(* IEC 61131-3 sources: POMIRTS_lab3/AS/Library/AsETH, 3 files *)

(* ---- AsETH.typ ---- *)
(********************************************************************
 * COPYRIGHT -- Bernecker + Rainer
 ********************************************************************
 * Library: AsEth
 * File: AsEth.typ
 * Author: B+R
 ********************************************************************
 * Data types of library AsEth
 ********************************************************************)

TYPE
    ethSTATISTICS_typ	: STRUCT				(*statistics*)
		bytesrecv		: UDINT;				(*bytes received*)
		bytessend		: UDINT;				(*bytes sent*)
		packetsrecv		: UDINT;				(*packets received*)
		packetssend		: UDINT;				(*packets send*)
		mcpacketsrecv	: UDINT;				(*multicast packets received*)
		mcpacketssend	: UDINT;				(*multicats packets sent*)
		errorrecv		: UDINT;				(*input errors*)
		errorsend		: UDINT;				(*output errors*)
		errorframe		: UDINT;				(*frame errors*)
		errorcrc		: UDINT;				(*crc errors*)
		collisions		: UDINT;				(*collisions*)
		latecollision	: UDINT;				(*late collisions*)
		drops			: UDINT;				(*dropped on input*)
		lostcarrier		: UDINT;				(*lost carrier*)
		underflow		: UDINT;				(*silo underflow*)
		retry			: UDINT;				(*retries after 16 collisions*)
		noproto			: UDINT;				(*destined for unsupported protocol*)
		intrecv			: UDINT;				(*reveive interrupts*)
		intsend			: UDINT;				(*transmit interrupts*)
		bufferrecv		: UDINT;				(*receive buffer errror*)
		buffersend		: UDINT;				(*send buffer errror*)
		broadcasts		: UDINT;				(*broadcasts*)
		broadcaststop	: UDINT;				(*broadcast stop*)
		reserve			: ARRAY[0..9] OF UDINT;	(*reserved for future use*)
	END_STRUCT;
END_TYPE

(* ---- AsETH.fun ---- *)
(********************************************************************
 * COPYRIGHT -- Bernecker + Rainer
 ********************************************************************
 * Library: AsEth
 * File: AsEth.fun
 * Author: B+R
 ********************************************************************
 * Functions and function blocks of library AsEth
 ********************************************************************)

FUNCTION_BLOCK EthStat					(*retrieves an interface's statistics; asynchronous execution*)
	VAR_INPUT
		enable			: BOOL;			(*enables execution*)
		pDevice			: UDINT;		(*device name given as a pointer*)
		pStat			: UDINT;		(*pointer to the statistic structure ethSTATISTICS_typ*)
	END_VAR

	VAR_OUTPUT
		status			: UINT;			(*execution status: ERR_OK, ERR_FUB_ENABLE_FALSE, ERR_FUB_BUSY, 0xXXXX = see help*)
	END_VAR

	VAR
        i_state			: UINT;			(*internal variable*)
		i_result		: UINT;			(*internal variable*)
        i_tmp			: UDINT;		(*internal variable*)
	END_VAR
END_FUNCTION_BLOCK

FUNCTION ethInetAton : UINT				(*converts an IP address from internet-format to binary value*)
	VAR_INPUT
		pIpStr		:UDINT;				(*address of the IP address (internet-format)*)
		pIpAdr		:UDINT;				(*address where to store the binary value (network order) of the IP address*)
	END_VAR
END_FUNCTION

FUNCTION ethInetNtoa : UINT				(*converts an IP address from binary value to internet-format*)
	VAR_INPUT
		ipAdr		:UDINT;				(*binary value (network order) of the IP address*)
		pIpStr		:UDINT;				(*address where to store the internet-format string of the IP address*)
	END_VAR
END_FUNCTION

(* ---- AsETH.var ---- *)
(********************************************************************
 * COPYRIGHT -- Bernecker + Rainer
 ********************************************************************
 * Library: AsEth
 * File: AsEth.var
 * Author: B+R
 ********************************************************************
 * Local variables of library AsEth
 ********************************************************************)

VAR CONSTANT
	ethERR_PARAMETER					: UINT := 32850;	(*invalid parameter, check parameter*)
	ethERR_SYSTEM						: UINT := 32899;	(*system error*)
END_VAR
